{attribute 'qualified_only'}
{attribute 'strict'}
TYPE E_SlitPairStatesV2 :
(
    eInit := 0,
    eEnableRealGenerators,
    eDisableRealGenerators,
    eEnableVirtualGenerators,
    eDisableVirtualGenerators,
    eWaitForVirtualMoveDone,
    eWaitForRealMoveDone,
    eError,
    eOperational,
    eWaitForVirtaulHomed,
    eWaitForRealHomed,
    eCheckRealAxisGeneratorsEnabled,
    eCheckVirtualAxisGeneratorsEnabled
);
END_TYPE

(* stored: Version 1.1.0.1, ProductVersion 3.1.4024.11
   DUT E_SlitPairStatesV2: Id {6665fbaf-b520-47d5-8ce7-9872d8af20f7} *)
